FUNCTION_BLOCK CU00xManualTask EXTENDS TcoTaskedService IMPLEMENTS ICUTask
VAR
END_VAR

Run();

(*~
	<docu>
		<summary>
			Main method of the sequener. Custom code needs to be placed here. The sequencer is executed by call of **Instance.Run()** method.
			This method is abstract, and it must be overridden in derived block.
		</summary>
	</docu>
~*)
METHOD PROTECTED Main : BOOL
Messenger.Notify('Running manual mode');
// Station.Components.OUT1.Service();
// Station.Components.OUT2.Service();
// Station.Components.OUT3.Service();
END_METHOD

METHOD PROTECTED OnStart
Station.AutomatTask.Restore();
Station.GroundTask.Restore();
Station.GroundTask.CancelGround();
END_METHOD

PROPERTY Station : REFERENCE TO CU00x
GET
VAR
    _station : POINTER TO CU00x;
END_VAR
IF __QUERYPOINTER(Parent, _station) THEN // Check if _Parent is Station001
    Station REF= _station^;              // If the check is successful dereference a pointer. simlar to THIS^ or SUPER^
END_IF
END_GET
END_PROPERTY

END_FUNCTION_BLOCK

(* stored: Version 1.1.0.1
   POU CU00xManualTask: Id {4da1dfbc-4c0a-47a8-95b6-4f0ca8024493}, SpecialFunc None
   Method Main: Id {b59a2119-19eb-4289-9c0b-227b833546df}
   Method OnStart: Id {9e5b3c71-1f5b-4076-a710-81816a9a4500}
   Property Station: Id {400a1f67-80cb-4f9f-a632-be597ac0ffc5}
   Get Get: Id {e3aceaef-61ff-438d-83cd-a8c6edd964ba} *)
